Staubli VAL3: onEdit.pgx

public program onEdit(string& x_sItem[])
  local string l_sItem
  local num l_nValue
  local string l_sType
  local bool l_bOk
begin
  //
  // compose the string
  call use:stringToArray(x_sItem,sItems)
  call getType(l_sType)
  //
  l_bOk=true
  toNum(sItems[1],l_nValue,l_bOk)
  // change the field
  call use:insertDialog(l_sType+" "+x_sItem+"#"+"DELAY [Sec] ",l_nValue,0,100)
  // give back
  x_sItem=sItems+","+toString(".2,",l_nValue)
end
